// TIA Portal project "3tank1havuzkarıştırıcı" (V20)

(* hardware
DEVICE "S7-1200 station_1"  S7-1200 Station
   slot 0: "Rack_0"  S7-1200 Rack  Rack  V1.0
   slot 1: "PLC_1"  CPU 1214C DC/DC/DC  6ES7 214-1AG40-0XB0  V4.7
*)

// ===== PLC "PLC_1"  CPU 1214C DC/DC/DC =====

VAR_GLOBAL   // PLC tag table "Default tag table"
   "Start but" AT %I0.0 : Bool;
   "Üst seviye sensörü 1" AT %I0.1 : Bool;
   "Üst seviye sensörü 2" AT %I0.2 : Bool;
   "Üst seviye sensörü 3" AT %I0.3 : Bool;
   "Alt seviye sensörü 1" AT %I0.4 : Bool;
   "Alt seviye sensörü 2" AT %I0.5 : Bool;
   "Alt seviye sensörü 3" AT %I0.6 : Bool;
   "Doldurma vanası 1" AT %Q0.0 : Bool;
   "Doldurma vanası 2" AT %Q0.1 : Bool;
   "Doldurma vanası 3" AT %Q0.2 : Bool;
   "Boşaltma vanası 1" AT %Q0.3 : Bool;
   "Boşaltma vanası 2" AT %Q0.4 : Bool;
   "Boşaltma vanası 3" AT %Q0.5 : Bool;
   "Isıtıcı 1" AT %Q0.6 : Bool;
   "Isıtıcı 2" AT %Q0.7 : Bool;
   "Isıtıcı 3" AT %Q1.0 : Bool;
   "Karıştırıcı" AT %Q1.1 : Bool;
   "kazan doldu mem" AT %M10.0 : Bool;
END_VAR

DATA_BLOCK "Isıtma ve karıştırma süreleri"   // DB1
{ S7_Optimized_Access := 'TRUE' }
VERSION : 0.1
   VAR
      "Kazan 1 ısıtma süresi" : Time := T#3s;
      "Kazan 2 ısıtma süresi" : Time := T#6s;
      "Kazan 3 ısıtma süresi" : Time := T#9s;
      "Karıştırma süresi" : Time := T#10s;
   END_VAR
BEGIN
END_DATA_BLOCK

DATA_BLOCK "Kazan 1"   // DB2
{ S7_Optimized_Access := 'TRUE' }
VERSION : 0.1
// stored: InstanceOfName Kazanlar
"Kazanlar"
BEGIN
END_DATA_BLOCK

DATA_BLOCK "Kazan 2"   // DB3
{ S7_Optimized_Access := 'TRUE' }
VERSION : 0.1
// stored: InstanceOfName Kazanlar
"Kazanlar"
BEGIN
END_DATA_BLOCK

DATA_BLOCK "Kazan 3"   // DB4
{ S7_Optimized_Access := 'TRUE' }
VERSION : 0.1
// stored: InstanceOfName Kazanlar
"Kazanlar"
BEGIN
END_DATA_BLOCK

// folder: System blocks/Program resources

DATA_BLOCK "timer 2"   // DB5
{ S7_Optimized_Access := 'TRUE' }
AUTHOR : Simatic
FAMILY : IEC
NAME : IEC_TMR
VERSION : 1.0
// stored: InstanceOfName IEC_TIMER
"IEC_TIMER"
BEGIN
END_DATA_BLOCK

// folder: (top level)

FUNCTION_BLOCK "Kazanlar"   // FB1, LAD
{ S7_Optimized_Access := 'TRUE' }
VERSION : 0.1
   VAR_INPUT
      Start : Bool;
      "Kazan dolu" : Bool;
      "Kazan boş" : Bool;
      "Isıtma süresi" : Time;
   END_VAR
   VAR_OUTPUT
      "Kazanı doldur" : Bool;
      "Kazanı boşalt" : Bool;
      "Isıtıcıyı çalıştır" : Bool;
   END_VAR
   VAR
      Merker1 : Bool;
      Merker3 : Bool;
      Merker2 : Bool;
      timer1 : TON_TIME;
   END_VAR
BEGIN

REGION Network 1
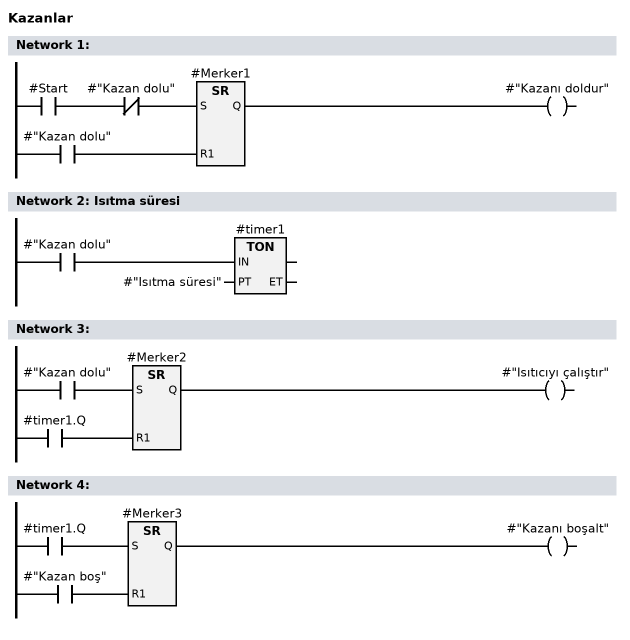
   RUNG wire#powerrail
      Contact( #Start )
      I_Contact( #"Kazan dolu" )
      S_SR(operand := #Merker1, r1 := wire#w1)
      Coil( #"Kazanı doldur" )
   END_RUNG
   RUNG wire#powerrail
      Contact( #"Kazan dolu" )
   END_RUNG wire#w1
   // the same network as SCL:
   IF #Start AND NOT #"Kazan dolu" THEN
       #Merker1 := TRUE;   // SR flip-flop
   END_IF;
   IF #"Kazan dolu" THEN #Merker1 := FALSE; END_IF;
   #"Kazanı doldur" := #Merker1;
END_REGION

REGION Network 2: Isıtma süresi
   #timer1(IN := #"Kazan dolu", PT := #"Isıtma süresi");   // TON
END_REGION

REGION Network 3
   RUNG wire#powerrail
      Contact( #"Kazan dolu" )
      S_SR(operand := #Merker2, r1 := wire#w1)
      Coil( #"Isıtıcıyı çalıştır" )
   END_RUNG
   RUNG wire#powerrail
      Contact( #timer1.Q )
   END_RUNG wire#w1
   // the same network as SCL:
   IF #"Kazan dolu" THEN
       #Merker2 := TRUE;   // SR flip-flop
   END_IF;
   IF #timer1.Q THEN #Merker2 := FALSE; END_IF;
   #"Isıtıcıyı çalıştır" := #Merker2;
END_REGION

REGION Network 4
   RUNG wire#powerrail
      Contact( #timer1.Q )
      S_SR(operand := #Merker3, r1 := wire#w1)
      Coil( #"Kazanı boşalt" )
   END_RUNG
   RUNG wire#powerrail
      Contact( #"Kazan boş" )
   END_RUNG wire#w1
   // the same network as SCL:
   IF #timer1.Q THEN
       #Merker3 := TRUE;   // SR flip-flop
   END_IF;
   IF #"Kazan boş" THEN #Merker3 := FALSE; END_IF;
   #"Kazanı boşalt" := #Merker3;
END_REGION
END_FUNCTION_BLOCK

ORGANIZATION_BLOCK "Main"   // OB1, LAD, ProgramCycle
TITLE = "Main Program Sweep (Cycle)"
{ S7_Optimized_Access := 'TRUE' }
VERSION : 0.1
   VAR_INPUT
      Initial_Call : Bool;   // Initial call of this OB
      Remanence : Bool;   // =True, if remanent data are available
   END_VAR
BEGIN

REGION Network 1
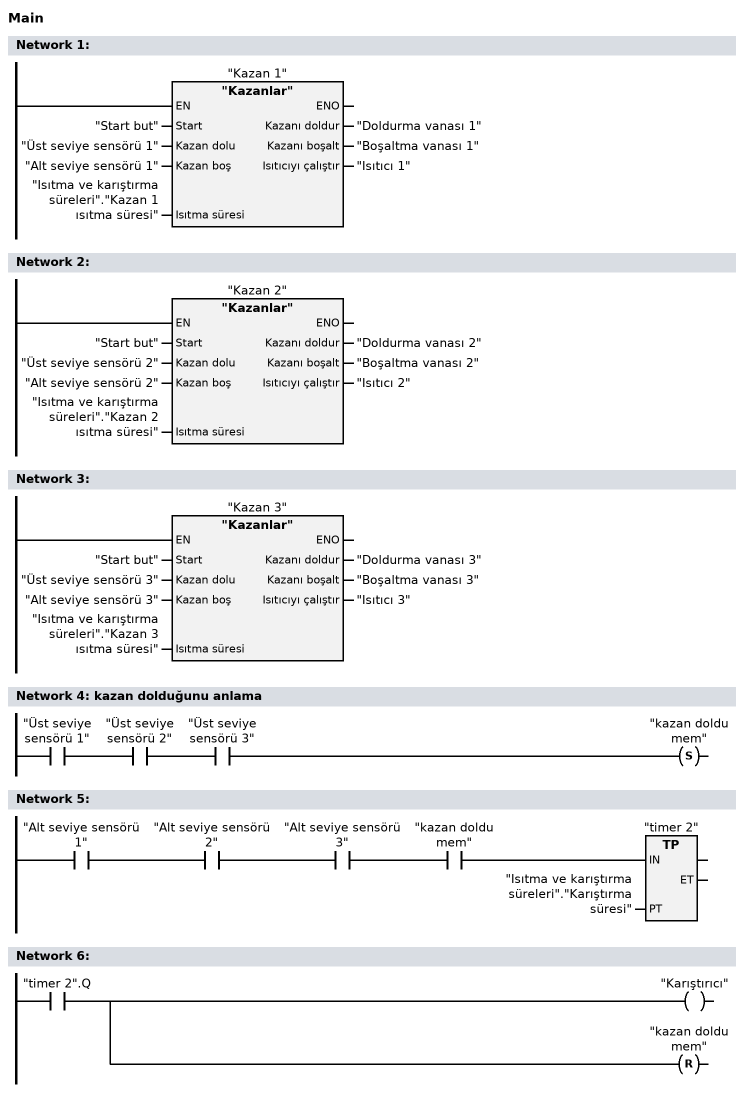
   RUNG wire#powerrail
      "Kazan 1"(Start := "Start but", "Kazan dolu" := "Üst seviye sensörü 1", "Kazan boş" := "Alt seviye sensörü 1", "Isıtma süresi" := "Isıtma ve karıştırma süreleri"."Kazan 1 ısıtma süresi", "Kazanı doldur" => "Doldurma vanası 1", "Kazanı boşalt" => "Boşaltma vanası 1", "Isıtıcıyı çalıştır" => "Isıtıcı 1")
   END_RUNG
   // the same network as SCL:
   "Kazan 1"(Start := "Start but",   // "Kazanlar"
             "Kazan dolu" := "Üst seviye sensörü 1",
             "Kazan boş" := "Alt seviye sensörü 1",
             "Isıtma süresi" := "Isıtma ve karıştırma süreleri"."Kazan 1 ısıtma süresi",
             "Kazanı doldur" => "Doldurma vanası 1",
             "Kazanı boşalt" => "Boşaltma vanası 1",
             "Isıtıcıyı çalıştır" => "Isıtıcı 1");
END_REGION

REGION Network 2
   RUNG wire#powerrail
      "Kazan 2"(Start := "Start but", "Kazan dolu" := "Üst seviye sensörü 2", "Kazan boş" := "Alt seviye sensörü 2", "Isıtma süresi" := "Isıtma ve karıştırma süreleri"."Kazan 2 ısıtma süresi", "Kazanı doldur" => "Doldurma vanası 2", "Kazanı boşalt" => "Boşaltma vanası 2", "Isıtıcıyı çalıştır" => "Isıtıcı 2")
   END_RUNG
   // the same network as SCL:
   "Kazan 2"(Start := "Start but",   // "Kazanlar"
             "Kazan dolu" := "Üst seviye sensörü 2",
             "Kazan boş" := "Alt seviye sensörü 2",
             "Isıtma süresi" := "Isıtma ve karıştırma süreleri"."Kazan 2 ısıtma süresi",
             "Kazanı doldur" => "Doldurma vanası 2",
             "Kazanı boşalt" => "Boşaltma vanası 2",
             "Isıtıcıyı çalıştır" => "Isıtıcı 2");
END_REGION

REGION Network 3
   RUNG wire#powerrail
      "Kazan 3"(Start := "Start but", "Kazan dolu" := "Üst seviye sensörü 3", "Kazan boş" := "Alt seviye sensörü 3", "Isıtma süresi" := "Isıtma ve karıştırma süreleri"."Kazan 3 ısıtma süresi", "Kazanı doldur" => "Doldurma vanası 3", "Kazanı boşalt" => "Boşaltma vanası 3", "Isıtıcıyı çalıştır" => "Isıtıcı 3")
   END_RUNG
   // the same network as SCL:
   "Kazan 3"(Start := "Start but",   // "Kazanlar"
             "Kazan dolu" := "Üst seviye sensörü 3",
             "Kazan boş" := "Alt seviye sensörü 3",
             "Isıtma süresi" := "Isıtma ve karıştırma süreleri"."Kazan 3 ısıtma süresi",
             "Kazanı doldur" => "Doldurma vanası 3",
             "Kazanı boşalt" => "Boşaltma vanası 3",
             "Isıtıcıyı çalıştır" => "Isıtıcı 3");
END_REGION

REGION Network 4: kazan dolduğunu anlama
   RUNG wire#powerrail
      Contact( "Üst seviye sensörü 1" )
      Contact( "Üst seviye sensörü 2" )
      Contact( "Üst seviye sensörü 3" )
      S_Coil( "kazan doldu mem" )
   END_RUNG
   // the same network as SCL:
   IF "Üst seviye sensörü 1" AND "Üst seviye sensörü 2" AND "Üst seviye sensörü 3" THEN
       "kazan doldu mem" := TRUE;
   END_IF;
END_REGION

REGION Network 5
   "timer 2".TP(IN := "Alt seviye sensörü 1" AND "Alt seviye sensörü 2" AND "Alt seviye sensörü 3" AND "kazan doldu mem",
                PT := "Isıtma ve karıştırma süreleri"."Karıştırma süresi");
END_REGION

REGION Network 6
   RUNG wire#powerrail
      Contact( "timer 2".Q )
      wire#w1
      Coil( "Karıştırıcı" )
   END_RUNG
   RUNG wire#w1
      R_Coil( "kazan doldu mem" )
   END_RUNG
   // the same network as SCL:
   "Karıştırıcı" := "timer 2".Q;
   IF "timer 2".Q THEN "kazan doldu mem" := FALSE; END_IF;
END_REGION
END_ORGANIZATION_BLOCK